FUNCTION TryConvert_ULINT_TO_BOOL : BOOL
VAR_INPUT
	in : ULINT;
	out : REFERENCE TO BOOL;
END_VAR

out := ULINT_TO_BOOL(in);
TryConvert_ULINT_TO_BOOL := TRUE;

END_FUNCTION

(* stored: Version 1.1.0.1, ProductVersion 3.1.4024.12
   POU TryConvert_ULINT_TO_BOOL: Id {123d1f1d-aa3e-420b-9308-c3eada0a1546}, SpecialFunc None *)
